Fanuc KAREL source: kd00035.KL

-- PROVISIONAL review KL for V1013-1; original PC SHA256 c59a2b653f4ee3c7992c6629802374f4bba04a9b4034322b531db068066e8bf3
-- Incomplete behavior may be omitted. Consult companion uncertainty JSON. Do not deploy.
PROGRAM KD00035
%NOLOCKGROUP
VAR
  I : INTEGER
  J : INTEGER
  B : BOOLEAN
  R : REAL
  S : STRING[80]
BEGIN
  -- UNRESOLVED_PC offsets 5-18; opcodes 9D,81,18,9D,1B,9D,12,9C,13,04
  -- UNRESOLVED_PC offsets 23-27; opcodes 7F
END KD00035
